Fanuc KAREL source: kt00739.KL

-- PROVISIONAL review KL for V940-1; original PC SHA256 36fc753e0337a6c1aa79d1b40a77d94d1ea55f2a88b04b59302ca359d09aed13
-- Incomplete behavior may be omitted. Consult companion uncertainty JSON. Do not deploy.
PROGRAM KT00739
%NOLOCKGROUP
VAR
  OUT : INTEGER
-- UNRESOLVED_DECL ARG type=002018
BEGIN
  -- V9_ZERO_TABLE_METADATA_HINT layout=0001; no indexed target words; source/name/runtime held
  -- UNRESOLVED_PC offsets 5-18; opcodes 22,1D,23
  -- UNRESOLVED_PC offsets 23-27; opcodes 7F
END KT00739
